FUNCTION_BLOCK EA_network2
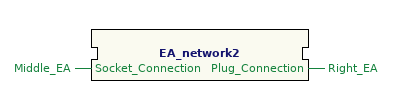
  SOCKETS
    Socket_Connection : Middle_EA;
  END_SOCKETS
  PLUGS
    Plug_Connection : Right_EA;
  END_PLUGS
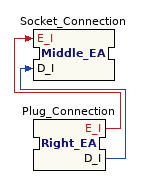
  EVENT_CONNECTIONS
    Plug_Connection.E_I TO Socket_Connection.E_I;
  END_CONNECTIONS
  DATA_CONNECTIONS
    Plug_Connection.D_I TO Socket_Connection.D_I;
  END_CONNECTIONS
END_FUNCTION_BLOCK
